TYPE T_MyType :
STRUCT
	a : UDINT;
	b : LREAL;
	c : STRING;
END_STRUCT
END_TYPE

(* stored: Version 1.1.0.1, ProductVersion 3.1.4024.12
   DUT T_MyType: Id {1df6c46d-2e8a-4dd5-9ea2-7ca6c2f6d59f} *)
